// TIA Portal V18 export
// export: Created 2026-06-08T17:17:40.7659824Z, ExportSetting WithDefaults, DisplayName Totally Integrated Automation Portal, DisplayVersion V18, DisplayName TIA Portal Openness, DisplayVersion V18, DisplayName TIA Portal Version Control Interface, DisplayVersion V18, DisplayName STEP 7 Professional, DisplayVersion V18, DisplayName STEP 7 Safety, DisplayVersion V18, DisplayName WinCC Professional, DisplayVersion V18
VAR_GLOBAL   // PLC tag table "Default tag table"
   L_LEVEL AT %I0.0 : Bool;
   H_LEVEL AT %I0.1 : Bool;
   STOP AT %I0.2 : Bool;
   PUMP_1 AT %Q0.0 : Bool;
   PUMP_2 AT %Q0.1 : Bool;
   VALVE AT %Q0.2 : Bool;
   MIXER AT %Q0.3 : Bool;
   Tag_2 AT %M0.0 : Bool;
   Tag_1 AT %M0.1 : Bool;
   Tag_3 AT %M0.2 : Bool;
END_VAR
